{attribute 'qualified_only'}
{attribute 'strict'}
TYPE MoverSequence :
(
	Off,
	Idle,
	MovingToStart,
	AtStart,
	MovingToStation,
	AtStation,
	Error,
	Stop,
	Stopping,
	RemoveAxes,
	RemovingAxes,
	Pausing,
	Paused,
	Disabling,
	Disabled,
	Waiting	
);
END_TYPE

(* stored: Version 1.1.0.1, ProductVersion 3.1.4026.8
   DUT MoverSequence: Id {222d4c05-bf8f-04c2-2b5f-d5019a5c0421} *)
